// TwinCAT 3 PLC project PLC
// ProgramVersion: 3.1.4024.0
// libraries:
//   Tc2_Standard, * (Beckhoff Automation GmbH)
//   Tc2_System, * (Beckhoff Automation GmbH)
//   Tc3_Module, * (Beckhoff Automation GmbH)
// project tree:
//   DUTs/ E_AutoMan.TcDUT, ST_CellConfig.TcDUT, ST_PartStatus.TcDUT
//   / GlobalTextList.TcGTLO, PlcTask.TcTTO
//   POUs/Cell/ E_CellState.TcDUT, FB_Cell.TcPOU
//   POUs/Devices/ FB_Axis.TcPOU, FB_Actuator.TcPOU, IActuator.TcIO, IAxis.TcIO
//   POUs/ MAIN.TcPOU
//   POUs/Stations/ E_StationState.TcDUT (not stored), FB_BarcodeScanner.TcPOU, FB_Filler.TcPOU, FB_Capper.TcPOU, FB_CheckWeigher.TcPOU, FB_Station.TcPOU, IStation.TcIO
// real-time tasks:
//   TASK PlcTask: cycle T#10ms, priority 20, ADS port 350
// variable links:
//   PLC/PLC Instance <-> SIM/SIM Instance
//     PlcTask Inputs/MAIN.fbCell.bPartPresentAtInfeed <-> PlcTask Outputs/MAIN.fbSimCell.bPartPresentAtInfeed
//     PlcTask Inputs/MAIN.fbCell.bPartPresentAtOutfeed <-> PlcTask Outputs/MAIN.fbSimCell.bPartPresentAtOutfeed
//     PlcTask Inputs/MAIN.fbCell.fbBarcoder.bPartPresent <-> PlcTask Outputs/MAIN.fbSimCell.fbSimScanner.bPartPresent
//     PlcTask Inputs/MAIN.fbCell.fbBarcoder.sBarcode <-> PlcTask Outputs/MAIN.fbSimCell.fbSimScanner.sBarcode
//     PlcTask Inputs/MAIN.fbCell.fbCapper.bCapDone <-> PlcTask Outputs/MAIN.fbSimCell.fbSimCapper.bCapDone
//     PlcTask Inputs/MAIN.fbCell.fbCapper.bCapFail <-> PlcTask Outputs/MAIN.fbSimCell.fbSimCapper.bCapFail
//     PlcTask Inputs/MAIN.fbCell.fbCapper.bPartPresent <-> PlcTask Outputs/MAIN.fbSimCell.fbSimCapper.bPartPresent
//     PlcTask Inputs/MAIN.fbCell.fbCheckWeigher.bPartPresent <-> PlcTask Outputs/MAIN.fbSimCell.fbSimWeigher.bPartPresent
//     PlcTask Inputs/MAIN.fbCell.fbCheckWeigher.fScaleReading <-> PlcTask Outputs/MAIN.fbSimCell.fbSimWeigher.fScaleReading
//     PlcTask Inputs/MAIN.fbCell.fbFiller.bPartPresent <-> PlcTask Outputs/MAIN.fbSimCell.fbSimFiller.bPartPresent
//     PlcTask Inputs/MAIN.fbCell.fbFiller.fVolumeFilled <-> PlcTask Outputs/MAIN.fbSimCell.fbSimFiller.fVolumeFilled
//     PlcTask Inputs/MAIN.fbCell.fbIndexConveyor.bBusy <-> PlcTask Outputs/MAIN.fbSimCell.fbIndexConveyor.bBusy
//     PlcTask Inputs/MAIN.fbCell.fbIndexConveyor.bError <-> PlcTask Outputs/MAIN.fbSimCell.fbIndexConveyor.bError
//     PlcTask Inputs/MAIN.fbCell.fbIndexConveyor.bReady <-> PlcTask Outputs/MAIN.fbSimCell.fbIndexConveyor.bReady
//     PlcTask Inputs/MAIN.fbCell.fbIndexConveyor.fActPosition <-> PlcTask Outputs/MAIN.fbSimCell.fbIndexConveyor.fActPosition
//     PlcTask Inputs/MAIN.fbCell.fbIndexConveyor.fActVelocity <-> PlcTask Outputs/MAIN.fbSimCell.fbIndexConveyor.fActVelocity
//     PlcTask Inputs/MAIN.fbCell.fbInfeedActuator.bExtended <-> PlcTask Outputs/MAIN.fbSimCell.fbInfeedActuator.bExtended
//     PlcTask Inputs/MAIN.fbCell.fbInfeedActuator.bRetracted <-> PlcTask Outputs/MAIN.fbSimCell.fbInfeedActuator.bRetracted
//     PlcTask Inputs/MAIN.fbCell.fbInfeedConveyor.bBusy <-> PlcTask Outputs/MAIN.fbSimCell.fbInfeedConveyor.bBusy
//     PlcTask Inputs/MAIN.fbCell.fbInfeedConveyor.bError <-> PlcTask Outputs/MAIN.fbSimCell.fbInfeedConveyor.bError
//     PlcTask Inputs/MAIN.fbCell.fbInfeedConveyor.bReady <-> PlcTask Outputs/MAIN.fbSimCell.fbInfeedConveyor.bReady
//     PlcTask Inputs/MAIN.fbCell.fbInfeedConveyor.fActPosition <-> PlcTask Outputs/MAIN.fbSimCell.fbInfeedConveyor.fActPosition
//     PlcTask Inputs/MAIN.fbCell.fbInfeedConveyor.fActVelocity <-> PlcTask Outputs/MAIN.fbSimCell.fbInfeedConveyor.fActVelocity
//     PlcTask Inputs/MAIN.fbCell.fbOutfeedActuator.bExtended <-> PlcTask Outputs/MAIN.fbSimCell.fbOutfeedActuator.bExtended
//     PlcTask Inputs/MAIN.fbCell.fbOutfeedActuator.bRetracted <-> PlcTask Outputs/MAIN.fbSimCell.fbOutfeedActuator.bRetracted
//     PlcTask Inputs/MAIN.fbCell.fbOutfeedConveyor.bBusy <-> PlcTask Outputs/MAIN.fbSimCell.fbOutfeedConveyor.bBusy
//     PlcTask Inputs/MAIN.fbCell.fbOutfeedConveyor.bError <-> PlcTask Outputs/MAIN.fbSimCell.fbOutfeedConveyor.bError
//     PlcTask Inputs/MAIN.fbCell.fbOutfeedConveyor.bReady <-> PlcTask Outputs/MAIN.fbSimCell.fbOutfeedConveyor.bReady
//     PlcTask Inputs/MAIN.fbCell.fbOutfeedConveyor.fActPosition <-> PlcTask Outputs/MAIN.fbSimCell.fbOutfeedConveyor.fActPosition
//     PlcTask Inputs/MAIN.fbCell.fbOutfeedConveyor.fActVelocity <-> PlcTask Outputs/MAIN.fbSimCell.fbOutfeedConveyor.fActVelocity
//     PlcTask Outputs/MAIN.fbCell.fFillRate <-> PlcTask Inputs/MAIN.fbSimCell.fFillRate
//     PlcTask Outputs/MAIN.fbCell.fbBarcoder.bTriggerRead <-> PlcTask Inputs/MAIN.fbSimCell.fbSimScanner.bTriggerRead
//     PlcTask Outputs/MAIN.fbCell.fbCapper.bCapTrigger <-> PlcTask Inputs/MAIN.fbSimCell.fbSimCapper.bCapTrigger
//     PlcTask Outputs/MAIN.fbCell.fbCapper.bClamp <-> PlcTask Inputs/MAIN.fbSimCell.fbSimCapper.bClamp
//     PlcTask Outputs/MAIN.fbCell.fbCheckWeigher.bLift <-> PlcTask Inputs/MAIN.fbSimCell.fbSimWeigher.bLift
//     PlcTask Outputs/MAIN.fbCell.fbFiller.bFillValve <-> PlcTask Inputs/MAIN.fbSimCell.fbSimFiller.bFillValve
//     PlcTask Outputs/MAIN.fbCell.fbIndexConveyor.bJogFwdCmd <-> PlcTask Inputs/MAIN.fbSimCell.fbIndexConveyor.bJogFwdCmd
//     PlcTask Outputs/MAIN.fbCell.fbIndexConveyor.bMoveAbsCmd <-> PlcTask Inputs/MAIN.fbSimCell.fbIndexConveyor.bMoveAbsCmd
//     PlcTask Outputs/MAIN.fbCell.fbIndexConveyor.fPositionCmd <-> PlcTask Inputs/MAIN.fbSimCell.fbIndexConveyor.fPositionCmd
//     PlcTask Outputs/MAIN.fbCell.fbIndexConveyor.fVelocityCmd <-> PlcTask Inputs/MAIN.fbSimCell.fbIndexConveyor.fVelocityCmd
//     PlcTask Outputs/MAIN.fbCell.fbInfeedActuator.bExtendCmd <-> PlcTask Inputs/MAIN.fbSimCell.fbInfeedActuator.bExtendCmd
//     PlcTask Outputs/MAIN.fbCell.fbInfeedActuator.bRetractCmd <-> PlcTask Inputs/MAIN.fbSimCell.fbInfeedActuator.bRetractCmd
//     PlcTask Outputs/MAIN.fbCell.fbInfeedConveyor.bJogFwdCmd <-> PlcTask Inputs/MAIN.fbSimCell.fbInfeedConveyor.bJogFwdCmd
//     PlcTask Outputs/MAIN.fbCell.fbInfeedConveyor.bMoveAbsCmd <-> PlcTask Inputs/MAIN.fbSimCell.fbInfeedConveyor.bMoveAbsCmd
//     PlcTask Outputs/MAIN.fbCell.fbInfeedConveyor.fPositionCmd <-> PlcTask Inputs/MAIN.fbSimCell.fbInfeedConveyor.fPositionCmd
//     PlcTask Outputs/MAIN.fbCell.fbInfeedConveyor.fVelocityCmd <-> PlcTask Inputs/MAIN.fbSimCell.fbInfeedConveyor.fVelocityCmd
//     PlcTask Outputs/MAIN.fbCell.fbOutfeedActuator.bExtendCmd <-> PlcTask Inputs/MAIN.fbSimCell.fbOutfeedActuator.bExtendCmd
//     PlcTask Outputs/MAIN.fbCell.fbOutfeedActuator.bRetractCmd <-> PlcTask Inputs/MAIN.fbSimCell.fbOutfeedActuator.bRetractCmd
//     PlcTask Outputs/MAIN.fbCell.fbOutfeedConveyor.bJogFwdCmd <-> PlcTask Inputs/MAIN.fbSimCell.fbOutfeedConveyor.bJogFwdCmd
//     PlcTask Outputs/MAIN.fbCell.fbOutfeedConveyor.bMoveAbsCmd <-> PlcTask Inputs/MAIN.fbSimCell.fbOutfeedConveyor.bMoveAbsCmd
//     PlcTask Outputs/MAIN.fbCell.fbOutfeedConveyor.fPositionCmd <-> PlcTask Inputs/MAIN.fbSimCell.fbOutfeedConveyor.fPositionCmd
//     PlcTask Outputs/MAIN.fbCell.fbOutfeedConveyor.fVelocityCmd <-> PlcTask Inputs/MAIN.fbSimCell.fbOutfeedConveyor.fVelocityCmd

CONFIGURATION PLC
    RESOURCE PLC ON TwinCAT3
        TASK PlcTask(INTERVAL := T#10ms, PRIORITY := 20);
        PROGRAM MAIN WITH PlcTask : MAIN;
    END_RESOURCE
END_CONFIGURATION

// ---- DUTs/E_AutoMan.TcDUT
{attribute 'qualified_only'}
{attribute 'strict'}
TYPE E_AutoMan :
(
	MANUAL := 0,
	AUTO := 1
);
END_TYPE

// ---- DUTs/ST_CellConfig.TcDUT
TYPE ST_CellConfig :
STRUCT
END_STRUCT
END_TYPE

// ---- DUTs/ST_PartStatus.TcDUT
TYPE ST_PartStatus :
STRUCT
	bBarcodeStatus			: BOOL := FALSE;
	sBarcode				: STRING(255) := '';
	bFillerStatus			: BOOL := FALSE;
	bCapperStatus			: BOOL := FALSE;
	bWeightStatus			: BOOL := FALSE;
	fActualWeightMg			: LREAL := 0.0;
END_STRUCT
END_TYPE

// ---- POUs/Cell/E_CellState.TcDUT
{attribute 'qualified_only'}
{attribute 'strict'}
TYPE E_CellState :
(
	STOPPED := 0,
	IDLE_WAIT := 1,
	FEED := 2,
	INDEX := 3
) DINT;
END_TYPE

// ---- POUs/Devices/IActuator.TcIO
INTERFACE IActuator

METHOD Cycle : BOOL
VAR_INPUT
END_VAR
END_METHOD

PROPERTY Error : BOOL
GET
END_GET
END_PROPERTY

METHOD Extend : BOOL
VAR_INPUT
END_VAR
END_METHOD

PROPERTY Extended : BOOL
GET
END_GET
END_PROPERTY

METHOD Retract : BOOL
VAR_INPUT
END_VAR
END_METHOD

PROPERTY Retracted : BOOL
GET
END_GET
END_PROPERTY

END_INTERFACE

// ---- POUs/Devices/IAxis.TcIO
INTERFACE IAxis

PROPERTY ActPosition : LREAL
GET
END_GET
END_PROPERTY

PROPERTY ActVelocity : LREAL
GET
END_GET
END_PROPERTY

PROPERTY Busy : BOOL
GET
END_GET
END_PROPERTY

METHOD Enable : BOOL
VAR_INPUT
END_VAR
END_METHOD

PROPERTY Enabled : BOOL
GET
END_GET
END_PROPERTY

PROPERTY Error : BOOL
GET
END_GET
END_PROPERTY

METHOD JogFwd : BOOL
VAR_INPUT
	Velocity		: LREAL;
END_VAR
END_METHOD

METHOD JogRev : BOOL
VAR_INPUT
	Velocity		: LREAL;
END_VAR
END_METHOD

METHOD MoveAbsolute : BOOL
VAR_INPUT
	Target		: LREAL;	// target position
	Velocity	: LREAL;
END_VAR
END_METHOD

METHOD Reset : BOOL
VAR_INPUT
END_VAR
END_METHOD

METHOD SetHome : BOOL
VAR_INPUT
	Target		: LREAL;
END_VAR
END_METHOD

METHOD StopMove : BOOL
VAR_INPUT
END_VAR
END_METHOD

END_INTERFACE

// ---- POUs/Stations/IStation.TcIO
INTERFACE IStation

METHOD Execute : PVOID
VAR_INPUT
END_VAR
END_METHOD

PROPERTY Faulted : BOOL
GET
END_GET
END_PROPERTY

PROPERTY PartPresent : BOOL
GET
END_GET
END_PROPERTY

PROPERTY PartStatus : POINTER TO ST_PartStatus
SET
END_SET
END_PROPERTY

PROPERTY Ready : BOOL
GET
END_GET
END_PROPERTY

END_INTERFACE

// ---- POUs/MAIN.TcPOU
PROGRAM MAIN
VAR
	fbCell 				: FB_Cell;
END_VAR

fbCell.Execute();

END_PROGRAM

// ---- POUs/Cell/FB_Cell.TcPOU
FUNCTION_BLOCK FB_Cell
VAR_INPUT
END_VAR
VAR_OUTPUT
END_VAR
VAR
	eAutoMan					: E_AutoMan := E_AutoMan.AUTO;
	State						: E_CellState;
	
	// IO
	bStartBtn					AT %I* : BOOL;
	bStopBtn					AT %I* : BOOL;
	bPartPresentAtInfeed		AT %I* : BOOL;
	bPartPresentAtOutfeed		AT %I* : BOOL;
	fFillRate					AT %Q* : LREAL := 2.5;
	
	// devices
	fbInfeedActuator			: FB_Actuator;
	fbOutfeedActuator			: FB_Actuator;
	fbInfeedConveyor			: FB_Axis;
	fbIndexConveyor				: FB_Axis;
	fbOutfeedConveyor			: FB_Axis;
	
	InfeedConveyor				: IAxis := fbInfeedConveyor;
	IndexConveyor				: IAxis := fbIndexConveyor;
	InfeedActuator				: IActuator := fbInfeedActuator;
	OutfeedActuator				: IActuator := fbOutfeedActuator;
	OutfeedConveyor				: IAxis := fbOutfeedConveyor;
	
	// stations
	fbBarcoder					: FB_BarcodeScanner;
	fbFiller					: FB_Filler;
	fbCapper					: FB_Capper;
	fbCheckWeigher				: FB_CheckWeigher;
	Stations					: ARRAY[0..3] OF IStation := [fbBarcoder, fbFiller, fbCapper, fbCheckWeigher];
	iStationCount				: DINT := 4;
	i							: DINT;
	
	bAllStationsReady			: BOOL;
	bCellPartPresent			: BOOL;
	bStationFaulted				: BOOL;
	tmrStationWait				: TON;
	bInFeeding					: BOOL;
	bIndexing					: BOOL;
	bOutfeeding					: BOOL;
	
	PartStatus					: ARRAY[0..3] OF ST_PartStatus;
	NewPart						: ST_PartStatus;
	OutfeedPart					: ST_PartStatus;
	
	fIndexPosition				: LREAL;
	INDEX_DIST					: LREAL := 300.0;
	INDEX_VEL					: LREAL := 100.0;
	INFEED_VEL					: LREAL := 100.0;
	
	bStartReq					: BOOL;
	bStopReq					: BOOL;
	bInit 						: BOOL := TRUE;
	
	bFillRateTest				: BOOL;
	tmrFillRate					: TON;
END_VAR

METHOD PRIVATE CheckPart : BOOL
VAR_INPUT
	Status			: ST_PartStatus;
END_VAR
CheckPart := Status.bBarcodeStatus AND Status.bFillerStatus AND Status.bCapperStatus AND Status.bWeightStatus;
END_METHOD

METHOD PUBLIC Execute : PVOID
StationMgr();

IF eAutoMan = E_AutoMan.AUTO THEN
	
	CASE State OF
		
		E_CellState.STOPPED:
			
			IF bStartReq THEN
				State := E_CellState.IDLE_WAIT;
				bStartReq := FALSE;
			END_IF
			
		E_CellState.IDLE_WAIT:
		
			IF bPartPresentAtInfeed AND Stations[0] <> 0 
			AND (Stations[0].Ready AND NOT Stations[0].PartPresent) THEN
				State := E_CellState.FEED;
			END_IF
			
			IF bAllStationsReady AND bCellPartPresent THEN
				tmrStationWait(IN:=TRUE, PT:=T#500MS);
				IF tmrStationWait.Q THEN
					tmrStationWait(IN:=FALSE);
					State := E_CellState.INDEX;
				END_IF
			END_IF
			
			IF bStopReq THEN
				State := E_CellState.STOPPED;
				bStopReq := FALSE;
			END_IF
			
		E_CellState.FEED:
		
			IF NOT bInFeeding THEN
				MEMCPY(ADR(PartStatus[0]), ADR(NewPart), SIZEOF(ST_PartStatus));
				bInFeeding := TRUE;
			END_IF
			
			IF InfeedActuator.Cycle() THEN
				State := E_CellState.IDLE_WAIT;
				bInFeeding := FALSE;
			END_IF
			
		E_CellState.INDEX:
			
			IF NOT bIndexing THEN
				fIndexPosition := IndexConveyor.ActPosition + INDEX_DIST;
				bIndexing := TRUE;
			END_IF
			
			IF (IndexConveyor.MoveAbsolute(fIndexPosition, INDEX_VEL)) AND bIndexing THEN
				bIndexing := FALSE;
				OutfeedPart := PartStatus[3];
				MEMCPY(ADR(PartStatus[1]), ADR(PartStatus[0]), SIZEOF(ST_PartStatus)*3);
				MEMSET(ADR(PartStatus[0]), 0, SIZEOF(ST_PartStatus));
				State := E_CellState.IDLE_WAIT;
			END_IF
			
	END_CASE
	
	IF State <> E_CellState.STOPPED THEN
		
		InfeedConveyor.JogFwd(INFEED_VEL);
		OutfeedConveyor.JogFwd(INFEED_VEL);
		
		IF bPartPresentAtOutfeed THEN
			// bad part
			IF NOT CheckPart(OutfeedPart) THEN
				bOutFeeding := TRUE;
			END_IF
		END_IF
		IF bOutfeeding THEN
			IF OutfeedActuator.Cycle() THEN
				bOutfeeding := FALSE;
			END_IF
		END_IF
		
		IF bFillRateTest THEN
			tmrFillRate(IN:=NOT tmrFillRate.Q, PT:=T#15M); 
			IF tmrFillRate.Q THEN
				fFillRate := fFillRate + 0.05;
			END_IF
		END_IF
		
	ELSE
		InfeedConveyor.StopMove();
		OutfeedConveyor.StopMove();
	END_IF
	
END_IF

IF bStartBtn THEN
	bStopReq := FALSE;
	bStartReq := TRUE;
END_IF

IF bStopBtn THEN
	bStartReq := FALSE;
	bStopReq := TRUE;
END_IF
END_METHOD

METHOD PRIVATE StationMgr : PVOID
VAR_INPUT
END_VAR
IF iStationCount < 1 THEN
	RETURN;
END_IF

IF bInit THEN
	FOR i:= 0 TO iStationCount - 1 DO
		Stations[i].PartStatus := ADR(PartStatus[i]);
	END_FOR
	bInit := FALSE;
END_IF

bAllStationsReady := TRUE;
bStationFaulted := FALSE;
bCellPartPresent := FALSE;

FOR i := 0 TO iStationCount - 1	DO
	IF (Stations[i] = 0) THEN
		CONTINUE;
	END_IF
	
	Stations[i].Execute();
	
	IF NOT Stations[i].Ready THEN
		bAllStationsReady := FALSE;
	END_IF
	
	IF Stations[i].Faulted THEN
		bStationFaulted := TRUE;
	END_IF
	
	IF Stations[i].PartPresent THEN
		bCellPartPresent := TRUE;
	END_IF
	
END_FOR
END_METHOD

END_FUNCTION_BLOCK

// ---- POUs/Devices/FB_Actuator.TcPOU
FUNCTION_BLOCK FB_Actuator IMPLEMENTS IActuator
VAR_INPUT
END_VAR
VAR_OUTPUT
END_VAR
VAR
	bExtended			AT %I* : BOOL;
	bRetracted			AT %I* : BOOL;
	bExtendCmd			AT %Q* : BOOL;
	bRetractCmd			AT %Q* : BOOL;
	
	iCycleState			: DINT;
	bError				: BOOL;
	tmrTimeout			: TON;
END_VAR

METHOD Cycle : BOOL
CASE iCycleState OF
	0:
		IF Extend() THEN
			iCycleState := 1;
		END_IF
	1:
		IF Retract() THEN
			iCycleState := 2;
		END_IF
		
	2:
		iCycleState := 0;
		Cycle := TRUE;
END_CASE
END_METHOD

PROPERTY Error : BOOL
GET
Error := bError;
END_GET
END_PROPERTY

METHOD Extend : BOOL
bRetractCmd := FALSE;
bExtendCmd := TRUE;
IF bExtended THEN
	bExtendCmd := FALSE;
	bError := FALSE;
	tmrTimeout(IN:=FALSE);
	Extend := TRUE;
ELSE
	tmrTimeout(IN:=TRUE, PT:=T#5S);
	IF tmrTimeout.Q THEN
		bError := TRUE;
	END_IF
END_IF
END_METHOD

PROPERTY Extended : BOOL
GET
Extended := bExtended;
END_GET
END_PROPERTY

METHOD Retract : BOOL
bExtendCmd := FALSE;
bRetractCmd := TRUE;
IF bRetracted THEN
	bRetractCmd := FALSE;
	bError := FALSE;
	tmrTimeout(IN:=FALSE);
	Retract := TRUE;
ELSE
	tmrTimeout(IN:=TRUE, PT:=T#5S);
	IF tmrTimeout.Q THEN
		bError := TRUE;
	END_IF
END_IF
END_METHOD

PROPERTY Retracted : BOOL
GET
Retracted := bRetracted;
END_GET
END_PROPERTY

END_FUNCTION_BLOCK

// ---- POUs/Devices/FB_Axis.TcPOU
FUNCTION_BLOCK FB_Axis IMPLEMENTS IAxis
VAR_INPUT
END_VAR
VAR_OUTPUT
END_VAR
VAR
	fActPosition			AT %I* : LREAL;
	fActVelocity			AT %I* : LREAL;
	bReady					AT %I* : BOOL;
	bBusy					AT %I* : BOOL;
	bError					AT %I* : BOOL;
	bRunning				AT %I* : BOOL;
	
	bJogFwdCmd				AT %Q* : BOOL;
	bMoveAbsCmd				AT %Q* : BOOL;
	fPositionCmd			AT %Q* : LREAL;
	fVelocityCmd			AT %Q* : LREAL;
	
	iMovCmdState			: DINT;
END_VAR

PROPERTY ActPosition : LREAL
GET
ActPosition := fActPosition;
END_GET
END_PROPERTY

PROPERTY ActVelocity : LREAL
GET
ActVelocity := fActVelocity;
END_GET
END_PROPERTY

PROPERTY Busy : BOOL
GET
Busy := bBusy;
END_GET
END_PROPERTY

METHOD Enable : BOOL
END_METHOD

PROPERTY Enabled : BOOL
GET
END_GET
END_PROPERTY

PROPERTY Error : BOOL
GET
Error := bError;
END_GET
END_PROPERTY

METHOD JogFwd : BOOL
VAR_INPUT
	Velocity	: LREAL;
END_VAR
fVelocityCmd := Velocity;
bJogFwdCmd := TRUE;
END_METHOD

METHOD JogRev : BOOL
VAR_INPUT
	Velocity	: LREAL;
END_VAR
END_METHOD

METHOD MoveAbsolute : BOOL
VAR_INPUT
	(* target position*)
	Target		: LREAL;
	Velocity	: LREAL;
END_VAR
fPositionCmd := Target;
fVelocityCmd := Velocity;

CASE iMovCmdState OF
	0:
		IF bReady THEN
			iMovCmdState := 1;
		END_IF
	1:
		bMoveAbsCmd := TRUE;
		IF bBusy THEN
			iMovCmdState := 2;
		END_IF	
	2:
		IF NOT bBusy THEN
			bMoveAbsCmd := FALSE;
			iMovCmdState := 0;
			MoveAbsolute := TRUE;
		END_IF
	
END_CASE
END_METHOD

METHOD Reset : BOOL
END_METHOD

METHOD SetHome : BOOL
VAR_INPUT
	Target	: LREAL;
END_VAR
END_METHOD

METHOD StopMove : BOOL
bJogFwdCmd := FALSE;
bMoveAbsCmd := FALSE;
END_METHOD

END_FUNCTION_BLOCK

// ---- POUs/Stations/FB_BarcodeScanner.TcPOU
FUNCTION_BLOCK FB_BarcodeScanner EXTENDS FB_Station
VAR_INPUT
END_VAR
VAR_OUTPUT
END_VAR
VAR
	bTriggerRead			AT %Q* : BOOL;
	sBarcode				AT %I* : STRING(255);
	
	sBarcodeRead			: STRING(255);
	iWorkState				: DINT;
	iRetries				: DINT;
	tmrRetry				: TON;
END_VAR
VAR CONSTANT
	NO_READ					: STRING(255) := 'NO_READ';
	READ_RETRY_COUNT		: DINT := 3;
END_VAR

METHOD PROTECTED  DoWork : BOOL
VAR_INPUT
END_VAR
CASE iWorkState OF
	0:
		iRetries := 0;
		sBarcodeRead := '';
		iWorkState := 10;
		bTriggerRead := TRUE;
		
	10:
		IF sBarcode <> '' THEN
			sBarcodeRead := sBarcode;
			bTriggerRead := FALSE;
			iWorkState := 20;
		END_IF
		
	11:
		tmrRetry(IN:=TRUE, PT:=T#500MS);
		IF tmrRetry.Q THEN
			tmrRetry(IN:=FALSE);
			bTriggerRead := TRUE;
			iWorkState := 10;
		END_IF
		
	20:
		IF sBarcodeRead = NO_READ THEN
			IF iRetries < READ_RETRY_COUNT THEN
				iRetries := iRetries + 1;
				iWorkState := 11;
			ELSE
				pPartStatus^.bBarcodeStatus := FALSE;
				pPartStatus^.sBarcode := NO_READ;
				iWorkState := 30;
			END_IF
		ELSE
			pPartStatus^.bBarcodeStatus := TRUE;
			pPartStatus^.sBarcode := sBarcodeRead;
			iWorkState := 30;
		END_IF
		
	30:
		iWorkState := 0;
		DoWork := TRUE;
	
END_CASE
END_METHOD

METHOD PROTECTED  FaultHandler : E_StationState
VAR_INPUT
END_VAR
END_METHOD

END_FUNCTION_BLOCK

// ---- POUs/Stations/FB_Station.TcPOU
FUNCTION_BLOCK ABSTRACT FB_Station IMPLEMENTS IStation
VAR_INPUT
END_VAR
VAR_OUTPUT
END_VAR
VAR
	bPartPresent			AT %I* : BOOL;
	bReady					: BOOL;
	bFaulted				: BOOL;
	bBusy					: BOOL;
	
	{attribute 'TcAnalytics'}
	eState					: E_StationState;
	pPartStatus				: POINTER TO ST_PartStatus;
	tmrPartPresentDelay		: TON;
END_VAR

METHOD PROTECTED ABSTRACT DoWork : BOOL
VAR_INPUT
END_VAR
END_METHOD

METHOD PUBLIC Execute : PVOID
bReady := NOT bFaulted AND NOT bBusy;

CASE eState OF
	
	E_StationState.IDLE_READY:
		
		tmrPartPresentDelay(IN:=bPartPresent, PT:=T#300MS);
		
		IF tmrPartPresentDelay.Q AND bReady THEN
			eState := E_StationState.PART_PRESENT;
		END_IF
	
	E_StationState.PART_PRESENT:
	
		bBusy := TRUE;
		eState := E_StationState.WORKING;
	
	E_StationState.WORKING:
	
		IF DoWork() THEN
			eState := E_StationState.WORK_COMPLETE;
		END_IF
		
		IF bFaulted THEN
			eState := E_StationState.FAULTED;
		END_IF
	
	E_StationState.WORK_COMPLETE:
		
		bBusy := FALSE;
		
		IF NOT bPartPresent THEN
			eState := E_StationState.IDLE_READY;
		END_IF
	
	E_StationState.FAULTED:
	
		eState := FaultHandler();

END_CASE
END_METHOD

PROPERTY Faulted : BOOL
GET
Faulted := bFaulted;
END_GET
END_PROPERTY

METHOD PROTECTED ABSTRACT FaultHandler : E_StationState
VAR_INPUT
END_VAR
END_METHOD

PROPERTY PartPresent : BOOL
GET
PartPresent := bPartPresent;
END_GET
END_PROPERTY

PROPERTY PartStatus : POINTER TO ST_PartStatus
SET
pPartStatus := PartStatus;
END_SET
END_PROPERTY

PROPERTY Ready : BOOL
GET
Ready := bReady;
END_GET
END_PROPERTY

PROPERTY State : E_StationState
GET
State := eState;
END_GET
END_PROPERTY

END_FUNCTION_BLOCK

// ---- POUs/Stations/FB_Filler.TcPOU
FUNCTION_BLOCK FB_Filler EXTENDS FB_Station
VAR_INPUT
END_VAR
VAR_OUTPUT
END_VAR
VAR
	fVolumeFilled			AT %I* : LREAL;
	bFillValve				AT %Q* : BOOL;
	
	fFillSetpoint			: LREAL := 1000.0;
	tmrDone					: TON;
	iWorkState				: DINT;
	
	fFillDoneDb				: LREAL := 1.0;
END_VAR

METHOD PROTECTED  DoWork : BOOL
VAR_INPUT
END_VAR
CASE iWorkState OF
	0:
		IF pPartStatus^.bBarcodeStatus THEN
			iWorkState := 10;
			bFillValve := TRUE;
		ELSE
			DoWork := TRUE;
		END_IF
		
		
	10:
		IF fVolumeFilled >= (fFillSetpoint - fFillDoneDb) THEN
			bFillValve := FALSE;
			pPartStatus^.bFillerStatus := TRUE;
			iWorkState := 20;
		END_IF
		
	20:
		tmrDone(IN:=TRUE, PT:=T#500MS);
		IF tmrDone.Q THEN
			tmrDone(IN:=FALSE);
			iWorkState := 0;
			DoWork := TRUE;
		END_IF
		
	
END_CASE
END_METHOD

METHOD PROTECTED  FaultHandler : E_StationState
VAR_INPUT
END_VAR
END_METHOD

PROPERTY PUBLIC FillSetpoint : LREAL
GET
FillSetpoint := fFillSetpoint;
END_GET
SET
fFillSetpoint := FillSetpoint;
END_SET
END_PROPERTY

END_FUNCTION_BLOCK

// ---- POUs/Stations/FB_Capper.TcPOU
FUNCTION_BLOCK FB_Capper EXTENDS FB_Station
VAR_INPUT
END_VAR
VAR_OUTPUT
END_VAR
VAR
	bClamp					AT %Q* : BOOL;
	bCapTrigger				AT %Q* : BOOL;
	bCapDone				AT %I* : BOOL;
	bCapFail				AT %I* : BOOL;
	
	tmrClamp				: TON;
	iWorkState				: DINT;
END_VAR
VAR CONSTANT
	CLAMP_TIME				: TIME := T#500MS;
END_VAR

METHOD PROTECTED  DoWork : BOOL
VAR_INPUT
END_VAR
CASE iWorkState OF
	0:
		IF pPartStatus^.bFillerStatus THEN
			bClamp := TRUE;
			tmrClamp(IN:=TRUE, PT:=CLAMP_TIME);
			IF tmrClamp.Q THEN
				tmrClamp(IN:=FALSE);
				iWorkState := 10;
			END_IF
		ELSE
			DoWork := TRUE;
		END_IF
		
		
	10:
		bCapTrigger := TRUE;
		IF bCapDone THEN
			iWorkState := 20; 
		END_IF
		
	20:
		bClamp := FALSE;
		tmrClamp(IN:=TRUE, PT:=CLAMP_TIME);
		IF tmrClamp.Q THEN
			tmrClamp(IN:=FALSE);
			pPartStatus^.bCapperStatus := NOT bCapFail;
			iWorkState := 30;
		END_IF
		
	30:
		bCapTrigger := FALSE;
		iWorkState := 0;
		DoWork := TRUE;
	
END_CASE
END_METHOD

METHOD PROTECTED  FaultHandler : E_StationState
VAR_INPUT
END_VAR
END_METHOD

END_FUNCTION_BLOCK

// ---- POUs/Stations/FB_CheckWeigher.TcPOU
FUNCTION_BLOCK FB_CheckWeigher EXTENDS FB_Station
VAR_INPUT
END_VAR
VAR_OUTPUT
END_VAR
VAR
	bLift					AT %Q* : BOOL;
	fScaleReading			AT %I* : LREAL;
	
	fWeightSetpoint			: LREAL := 1000;
	iWorkState				: DINT;
	tmrLift					: TON;
	tmrWeigh				: TON;
END_VAR
VAR CONSTANT
	WEIGH_DB_HI				: LREAL := 1.0;
	WEIGH_DB_LO				: LREAL := 0.2;
END_VAR

METHOD PROTECTED  DoWork : BOOL
VAR_INPUT
END_VAR
CASE iWorkState OF
	0:
		IF pPartStatus^.bCapperStatus THEN
			bLift := TRUE;
			tmrLift(IN:=TRUE, PT:=T#500MS);
			IF tmrLift.Q THEN
				tmrLift(IN:=FALSE);
				iWorkState := 10;
			END_IF
		ELSE
			DoWork := TRUE;
		END_IF
		
		
	10:
		tmrWeigh(IN:=TRUE, PT:=T#2S);
		IF tmrWeigh.Q THEN
			tmrWeigh(IN:=FALSE);
			pPartStatus^.fActualWeightMg := fScaleReading;
			iWorkState := 20;
		END_IF
		
	20:
		pPartStatus^.bWeightStatus := (pPartStatus^.fActualWeightMg > fWeightSetpoint - WEIGH_DB_LO)
			AND (pPartStatus^.fActualWeightMg < fWeightSetpoint + WEIGH_DB_HI);
		iWorkState := 30;
		
	30:
		bLift := FALSE;
		iWorkState := 0;
		DoWork := TRUE;
	
END_CASE
END_METHOD

METHOD PROTECTED  FaultHandler : E_StationState
VAR_INPUT
END_VAR
END_METHOD

PROPERTY WeightSetpoint : LREAL
GET
WeightSetpoint := fWeightSetpoint;
END_GET
SET
fWeightSetpoint := WeightSetpoint;
END_SET
END_PROPERTY

END_FUNCTION_BLOCK

// ---- GlobalTextList.TcGTLO
TEXTLIST GlobalTextList
  448 = 'Start'
END_TEXTLIST
